TYPE LogStruct :
STRUCT
	sales : REAL;
END_STRUCT
END_TYPE

(* stored: Version 1.1.0.1, ProductVersion 3.1.4024.10
   DUT LogStruct: Id {7cae65f2-b6d2-4340-81ff-d7c567d8a452} *)
